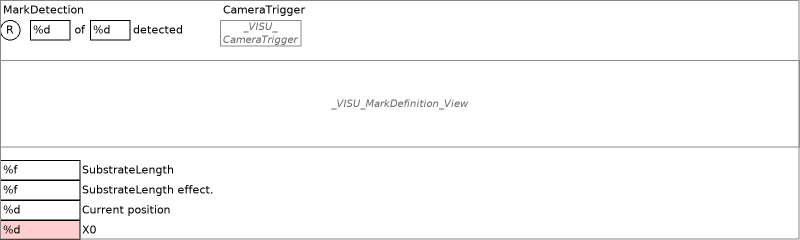
VISUALIZATION _VISU_MarkDetection  // 800x240
VAR_IN_OUT
	mInst: FB_MarkDetection;
END_VAR
    Rectangle (0,0 120x20), "MarkDetection"
    Rectangle (90,20 40x20), "%d", tooltip "teached marks", text variable: mInst._pFbMarkDefinition^._nMarks
    Rectangle (30,20 40x20), "%d", tooltip "detected marks", text variable: mInst._pFbMarkDefinition^._nMarksDetected, colour toggle: mInst._pFbMarkDefinition^._nMarksDetected >= mInst._pFbMarkDefinition^._nMarks AND mInst._pFbMarkDefinition^._nMarks > 0
    Ellipse (0,20 20x20), "R", tooltip "Reset"
        tap mInst.bManualReset
    Frame (220,20 81x26)
        shows _VISU_CameraTrigger(mInst := mInst)
    Rectangle (220,0 120x20), "CameraTrigger"
    Rectangle (130,20 60x20), "detected"
    Rectangle (70,20 20x20), "of"
    Rectangle (0,160 80x20), "%f", text variable: mInst._fSubstrateLength
    Rectangle (79,160 140x20), "SubstrateLength"
    Rectangle (0,180 80x20), "%f", text variable: mInst._fSubstrateLength
    Rectangle (79,180 140x20), "SubstrateLength effect."
    Rectangle (0,220 80x20), "%d", text variable: mInst._nX0, colour toggle: mInst._bValid
    Rectangle (79,220 140x20), "X0"
    Rectangle (0,200 80x20), "%d", text variable: mInst.nCurrentPos
    Rectangle (79,200 140x20), "Current position"
    Frame (0,60 800x87)
        shows _VISU_MarkDefinition_View(mInst := mInst._pFbMarkDefinition^, xScale := mInst.nMarkXMoveScale)
END_VISUALIZATION

(* stored: Version 1.1.0.1, ProductVersion 3.1.4024.11
   Visu _VISU_MarkDetection: Id {2576b8fd-c456-4caf-be04-cc964429f67a} *)
